Fanuc KAREL source: kt00040.KL

-- PROVISIONAL review KL for V1013-1; original PC SHA256 ef92799431b1b304a5250866008a5d58aa60218979a8bda0699a6ad0458ecc82
-- Incomplete behavior may be omitted. Consult companion uncertainty JSON. Do not deploy.
PROGRAM KT00040
%NOLOCKGROUP
VAR
  I1 : INTEGER
  OUT : REAL
-- UNRESOLVED_DECL H2 type=002017
BEGIN
  -- UNRESOLVED_PC offsets 5-16; opcodes 2E,23
  -- UNRESOLVED_PC offsets 21-35; opcodes 2E,22,9D,33,B4
  -- UNRESOLVED_PC offsets 40-63; opcodes 21,22,9D,33,B3,53,64,23
  -- UNRESOLVED_PC offsets 68-72; opcodes 7F
END KT00040
